Fanuc KAREL source: kt00586.KL

-- PROVISIONAL review KL for V1013-1; original PC SHA256 987837d0af2b88a0f94afa04105016f276429d8f1d67327a16086a3697dd17cb
-- Incomplete behavior may be omitted. Consult companion uncertainty JSON. Do not deploy.
PROGRAM KT00586
%NOLOCKGROUP
VAR
  I1 : INTEGER
-- UNRESOLVED_DECL V2 type=000013
-- UNRESOLVED_DECL OUT type=000013
BEGIN
  -- UNRESOLVED_PC offsets 5-16; opcodes 2E,23
  -- UNRESOLVED_PC offsets 21-36; opcodes 2E,22,32,35
  -- UNRESOLVED_PC offsets 41-63; opcodes 21,49,8F,4A
  -- UNRESOLVED_PC offsets 68-72; opcodes 7F
END KT00586
